// TIA Portal project "FactoryIO_Template_S7-1200_V16_V16" (V16)
// Vorlageprojekt für das Buch mit Zielsystem S7-1200

(* hardware
DEVICE "S7-1200-Station_1"  S7-1200 Station
   slot 0: "Baugruppenträger_0"  Rack  V1.0
   slot 1: "PLC_1"  CPU 1211C DC/DC/DC  6ES7 211-1AE40-0XB0  V4.1
*)

// ===== PLC "PLC_1"  CPU 1211C DC/DC/DC =====

VAR_GLOBAL   // PLC tag table "Standard-Variablentabelle"
   "Tag_4" AT %I10.0 : Bool;
   "Tag_5" AT %Q10.0 : Bool;
   "Tag_6" AT %I10.1 : Bool;
   "loop marker" AT %M0.0 : Bool;
   "Before Two Axis (-)" AT %M0.1 : Bool;
   "Tag_1" AT %M2.0 : Bool;
   "Tag_2" AT %M2.1 : Bool;
   "Tag_3" AT %M2.2 : Bool;
   "Tag_7" AT %M2.3 : Bool;
   "z-move-s1" AT %M0.2 : Bool;
   "stop x -s1" AT %M0.3 : Bool;
   "x-move-s1" AT %M0.4 : Bool;
   "rotate CC-1" AT %M0.5 : Bool;
   "rotate CCW-1" AT %M0.6 : Bool;
   "x-move-s2" AT %M0.7 : Bool;
   "z-move-s2" AT %M1.0 : Bool;
   "stop x -s2" AT %M1.1 : Bool;
   "counter reset marker" AT %M1.2 : Bool;
   "grab control" AT %M1.3 : Bool;
END_VAR

VAR_GLOBAL   // PLC tag table "Tag table from XML_1"
   "Start Button" AT %I0.0 : Bool;
   "Stop Button" AT %I0.1 : Bool;
   "low sensor" AT %I0.2 : Bool;
   "High Sensor" AT %I0.3 : Bool;
   "Before Two Axis" AT %I0.4 : Bool;
   "Two-Axis Pick & Place  (Moving X Detected)" AT %I0.5 : Bool;
   "Two-Axis Pick & Place  (Moving Z Detected)" AT %I0.6 : Bool;
   "Two-Axis Pick & Place  (Detected)" AT %I0.7 : Bool;
   "Two-Axis Pick & Place  (Rotating Detected)" AT %I1.0 : Bool;
   "Entry Conveyor" AT %Q0.0 : Bool;
   "Sorting Conveyor" AT %Q0.1 : Bool;
   "Small Conveyor" AT %Q0.2 : Bool;
   "Large Conveyor" AT %Q0.3 : Bool;
   "Two-Axis Pick & Place  (Moving X)" AT %Q0.4 : Bool;
   "Two-Axis Pick & Place  (Moving Z)" AT %Q0.5 : Bool;
   "Two-Axis Pick & Place  (Grab)" AT %Q0.6 : Bool;
   "Two-Axis Pick & Place  (Rotate CW)" AT %Q0.7 : Bool;
   "Two-Axis Pick & Place  (Rotate CCW)" AT %Q1.0 : Bool;
   "Start Button  (Light)" AT %Q1.1 : Bool;
   "Stop Button  (Light)" AT %Q1.2 : Bool;
END_VAR

// folder: System blocks/Program resources

DATA_BLOCK "movement-counter"   // DB1
{ S7_Optimized_Access := 'TRUE' }
AUTHOR : Simatic
FAMILY : IEC
NAME : CNTR
VERSION : 1.0
// stored: InstanceOfName IEC_COUNTER
"IEC_COUNTER"
BEGIN
END_DATA_BLOCK

DATA_BLOCK "grap-delay"   // DB2
{ S7_Optimized_Access := 'TRUE' }
AUTHOR : Simatic
FAMILY : IEC
NAME : IEC_TMR
VERSION : 1.0
// stored: InstanceOfName IEC_TIMER
"IEC_TIMER"
BEGIN
END_DATA_BLOCK

DATA_BLOCK "release delay"   // DB3
{ S7_Optimized_Access := 'TRUE' }
AUTHOR : Simatic
FAMILY : IEC
NAME : IEC_TMR
VERSION : 1.0
// stored: InstanceOfName IEC_TIMER
"IEC_TIMER"
BEGIN
END_DATA_BLOCK

// folder: (top level)

FUNCTION "MHJ-PLC-Lab-Function-S71200" : Void   // FC9000, SCL
{ S7_Optimized_Access := 'TRUE' }
VERSION : 0.1
   VAR_TEMP
      rdTimeReturn : Int;
      outputTime : DTL;
      SyncVal : Byte;
      forVal : Int;
      forVal_2 : Int;
      Value : Byte;
   END_VAR
   VAR CONSTANT
      CompVal : Byte := 16#34;
      Value_01 : Byte := 16#11;
      Value_01_DW : DWord := 16#A165_D992;
      Value_02_DW : DWord := 16#58BE_4401;
   END_VAR
BEGIN

   #Value:=PEEK(area := 16#82,
        dbNumber := 0,
        byteOffset := 511);
   #Value := #Value + 1;

   POKE(area := 16#82,
        dbNumber := 0,
        byteOffset := 511,
        value := #Value);

   POKE(area:=16#81,
        dbNumber:=0,
        byteOffset:=1016,
        value:=#Value_01_DW);
   POKE(area := 16#81,
        dbNumber := 0,
        byteOffset := 1020,
        value := #Value_02_DW);

   POKE(area := 16#81,
        dbNumber := 0,
        byteOffset := 511,
        value := B#16#00);

   FOR #forVal := 0 TO 120 DO
       FOR #forVal_2:=0 TO 10 DO
           #rdTimeReturn:=RD_SYS_T(#outputTime);
           #rdTimeReturn := WR_SYS_T(#outputTime);
           #rdTimeReturn := RD_SYS_T(#outputTime);
           #rdTimeReturn := WR_SYS_T(#outputTime);
       END_FOR;
       #SyncVal:= PEEK(area := 16#81,
                      dbNumber := 0,
                      byteOffset := 511);
       IF #SyncVal = #CompVal THEN
          GOTO M_1;
       END_IF;
   END_FOR;
   RETURN;

   M_1:
   POKE(area := 16#81,
        dbNumber := 0,
        byteOffset := 511,
        value := B#16#0);
END_FUNCTION

ORGANIZATION_BLOCK "Main"   // OB1, LAD, ProgramCycle
TITLE = "Main Program Sweep (Cycle)"
{ S7_Optimized_Access := 'TRUE' }
VERSION : 0.1
   VAR_INPUT
      Initial_Call : Bool;   // Initial call of this OB
      Remanence : Bool;   // =True, if remanent data are available
   END_VAR
   VAR_TEMP   // added for the SCL form of the ladder/FBD networks
      _w1 : Bool;
      _w2 : Bool;
      _w3 : Bool;
   END_VAR
BEGIN

REGION Network 1: Konnektierungsbaustein für PLC-Lab
   // Im Netzwerk 1 wird der Konnektierungsbaustein für PLC-Lab aufgerufen.
   // Dieser Aufruf darf nicht entfernt werden!
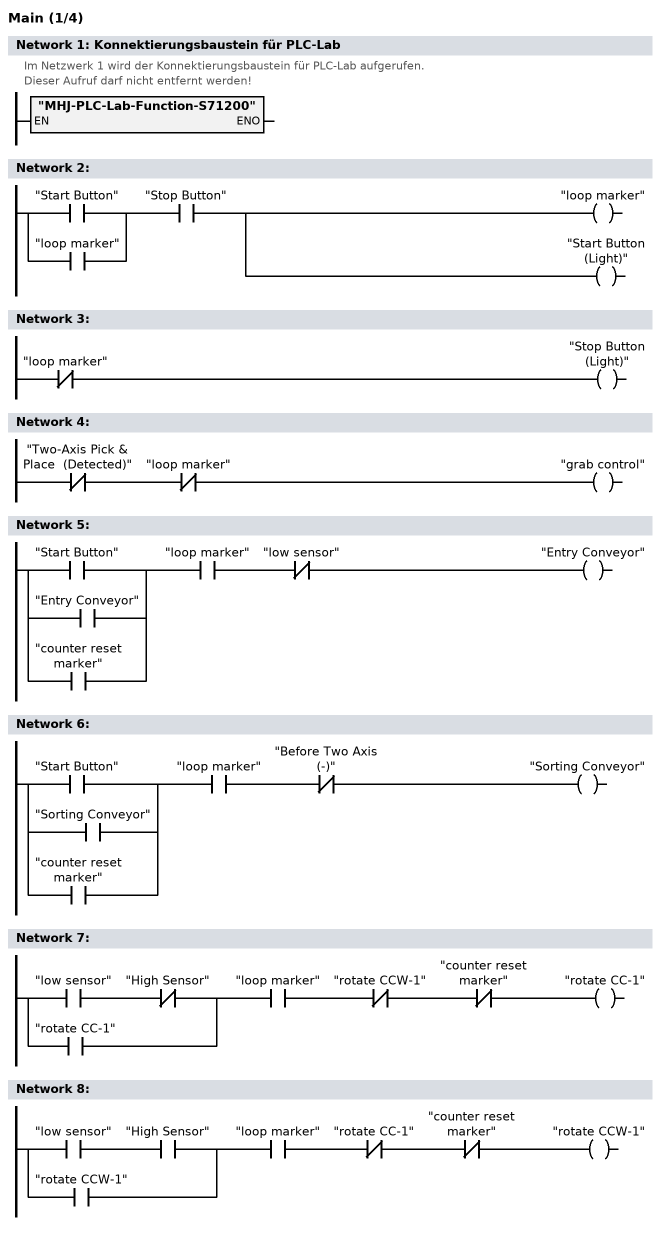
   RUNG wire#powerrail
      "MHJ-PLC-Lab-Function-S71200"()
   END_RUNG
   // the same network as SCL:
   "MHJ-PLC-Lab-Function-S71200"();
END_REGION

REGION Network 2
   RUNG wire#powerrail
      Contact( "Start Button" )
      wire#w1
      Contact( "Stop Button" )
      wire#w2
      Coil( "loop marker" )
   END_RUNG
   RUNG wire#powerrail
      Contact( "loop marker" )
   END_RUNG wire#w1
   RUNG wire#w2
      Coil( "Start Button  (Light)" )
   END_RUNG
   // the same network as SCL:
   "loop marker" := ("Start Button" OR "loop marker") AND "Stop Button";
   "Start Button  (Light)" := "loop marker";
END_REGION

REGION Network 3
   RUNG wire#powerrail
      I_Contact( "loop marker" )
      Coil( "Stop Button  (Light)" )
   END_RUNG
   // the same network as SCL:
   "Stop Button  (Light)" := NOT "loop marker";
END_REGION

REGION Network 4
   RUNG wire#powerrail
      I_Contact( "Two-Axis Pick & Place  (Detected)" )
      I_Contact( "loop marker" )
      Coil( "grab control" )
   END_RUNG
   // the same network as SCL:
   "grab control" := NOT "Two-Axis Pick & Place  (Detected)" AND NOT "loop marker";
END_REGION

REGION Network 5
   RUNG wire#powerrail
      Contact( "Start Button" )
      wire#w1
      Contact( "loop marker" )
      I_Contact( "low sensor" )
      Coil( "Entry Conveyor" )
   END_RUNG
   RUNG wire#powerrail
      Contact( "Entry Conveyor" )
   END_RUNG wire#w1
   RUNG wire#powerrail
      Contact( "counter reset marker" )
   END_RUNG wire#w1
   // the same network as SCL:
   "Entry Conveyor" := ("Start Button" OR "Entry Conveyor" OR "counter reset marker") AND "loop marker" AND NOT "low sensor";
END_REGION

REGION Network 6
   RUNG wire#powerrail
      Contact( "Start Button" )
      wire#w1
      Contact( "loop marker" )
      I_Contact( "Before Two Axis (-)" )
      Coil( "Sorting Conveyor" )
   END_RUNG
   RUNG wire#powerrail
      Contact( "Sorting Conveyor" )
   END_RUNG wire#w1
   RUNG wire#powerrail
      Contact( "counter reset marker" )
   END_RUNG wire#w1
   // the same network as SCL:
   "Sorting Conveyor" := ("Start Button" OR "Sorting Conveyor" OR "counter reset marker") AND "loop marker" AND NOT "Before Two Axis (-)";
END_REGION

REGION Network 7
   RUNG wire#powerrail
      Contact( "low sensor" )
      I_Contact( "High Sensor" )
      wire#w1
      Contact( "loop marker" )
      I_Contact( "rotate CCW-1" )
      I_Contact( "counter reset marker" )
      Coil( "rotate CC-1" )
   END_RUNG
   RUNG wire#powerrail
      Contact( "rotate CC-1" )
   END_RUNG wire#w1
   // the same network as SCL:
   "rotate CC-1" := (("low sensor" AND NOT "High Sensor") OR "rotate CC-1") AND "loop marker" AND NOT "rotate CCW-1" AND NOT "counter reset marker";
END_REGION

REGION Network 8
   RUNG wire#powerrail
      Contact( "low sensor" )
      Contact( "High Sensor" )
      wire#w1
      Contact( "loop marker" )
      I_Contact( "rotate CC-1" )
      I_Contact( "counter reset marker" )
      Coil( "rotate CCW-1" )
   END_RUNG
   RUNG wire#powerrail
      Contact( "rotate CCW-1" )
   END_RUNG wire#w1
   // the same network as SCL:
   "rotate CCW-1" := (("low sensor" AND "High Sensor") OR "rotate CCW-1") AND "loop marker" AND NOT "rotate CC-1" AND NOT "counter reset marker";
END_REGION

REGION Network 9
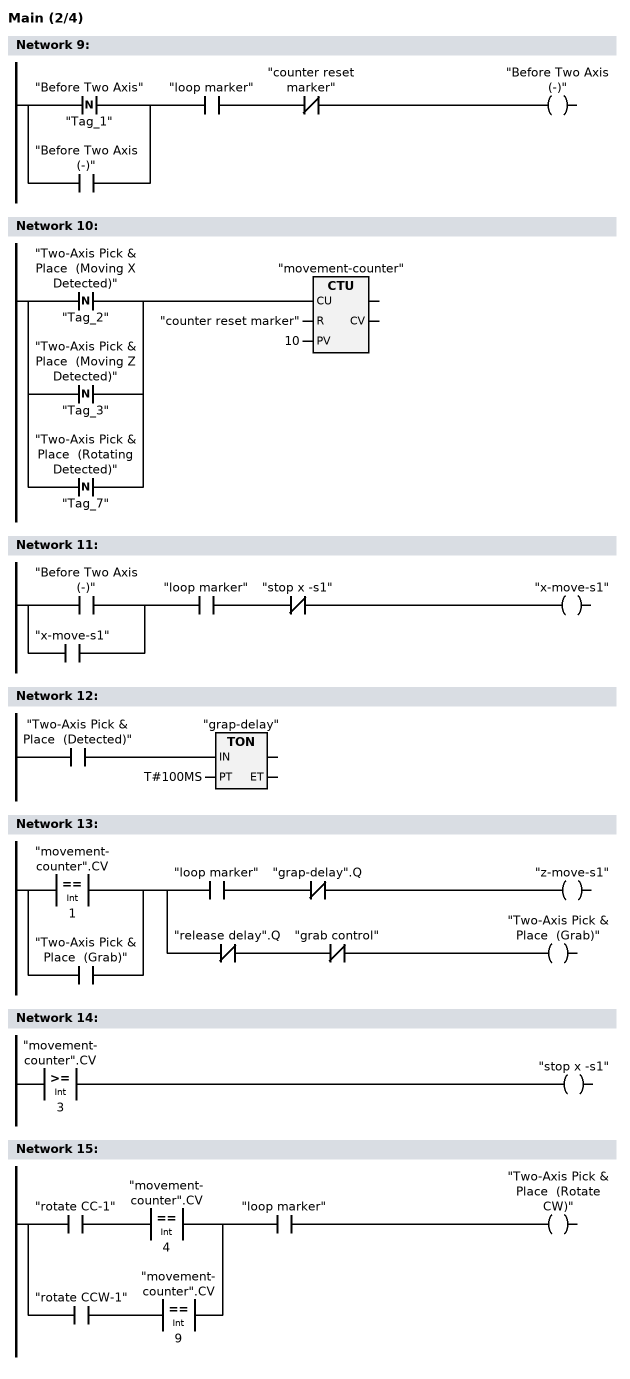
   RUNG wire#powerrail
      N_Contact(operand := "Before Two Axis", bit := "Tag_1")
      wire#w1
      Contact( "loop marker" )
      I_Contact( "counter reset marker" )
      Coil( "Before Two Axis (-)" )
   END_RUNG
   RUNG wire#powerrail
      Contact( "Before Two Axis (-)" )
   END_RUNG wire#w1
   // the same network as SCL:
   #_w1 := NOT "Before Two Axis" AND "Tag_1";   // falling edge of "Before Two Axis"
   "Tag_1" := "Before Two Axis";
   "Before Two Axis (-)" := (#_w1 OR "Before Two Axis (-)") AND "loop marker" AND NOT "counter reset marker";
END_REGION

REGION Network 10
   #_w1 := NOT "Two-Axis Pick & Place  (Moving X Detected)" AND "Tag_2";   // falling edge of "Two-Axis Pick & Place  (Moving X Detected)"
   "Tag_2" := "Two-Axis Pick & Place  (Moving X Detected)";
   #_w2 := NOT "Two-Axis Pick & Place  (Moving Z Detected)" AND "Tag_3";   // falling edge of "Two-Axis Pick & Place  (Moving Z Detected)"
   "Tag_3" := "Two-Axis Pick & Place  (Moving Z Detected)";
   #_w3 := NOT "Two-Axis Pick & Place  (Rotating Detected)" AND "Tag_7";   // falling edge of "Two-Axis Pick & Place  (Rotating Detected)"
   "Tag_7" := "Two-Axis Pick & Place  (Rotating Detected)";
   "movement-counter".CTU(CU := #_w1 OR #_w2 OR #_w3, R := "counter reset marker", PV := 10);
END_REGION

REGION Network 11
   RUNG wire#powerrail
      Contact( "Before Two Axis (-)" )
      wire#w1
      Contact( "loop marker" )
      I_Contact( "stop x -s1" )
      Coil( "x-move-s1" )
   END_RUNG
   RUNG wire#powerrail
      Contact( "x-move-s1" )
   END_RUNG wire#w1
   // the same network as SCL:
   "x-move-s1" := ("Before Two Axis (-)" OR "x-move-s1") AND "loop marker" AND NOT "stop x -s1";
END_REGION

REGION Network 12
   "grap-delay".TON(IN := "Two-Axis Pick & Place  (Detected)", PT := T#100MS);
END_REGION

REGION Network 13
   RUNG wire#powerrail
      { S7_Templates := "SrcType := Int" } EQ_Contact(in1 := "movement-counter".CV, in2 := 1)
      wire#w1
      Contact( "loop marker" )
      I_Contact( "grap-delay".Q )
      Coil( "z-move-s1" )
   END_RUNG
   RUNG wire#powerrail
      Contact( "Two-Axis Pick & Place  (Grab)" )
   END_RUNG wire#w1
   RUNG wire#w1
      I_Contact( "release delay".Q )
      I_Contact( "grab control" )
      Coil( "Two-Axis Pick & Place  (Grab)" )
   END_RUNG
   // the same network as SCL:
   #_w1 := ("movement-counter".CV = 1) OR "Two-Axis Pick & Place  (Grab)";
   "z-move-s1" := #_w1 AND "loop marker" AND NOT "grap-delay".Q;
   "Two-Axis Pick & Place  (Grab)" := #_w1 AND NOT "release delay".Q AND NOT "grab control";
END_REGION

REGION Network 14
   RUNG wire#powerrail
      { S7_Templates := "SrcType := Int" } GE_Contact(in1 := "movement-counter".CV, in2 := 3)
      Coil( "stop x -s1" )
   END_RUNG
   // the same network as SCL:
   "stop x -s1" := "movement-counter".CV >= 3;
END_REGION

REGION Network 15
   RUNG wire#powerrail
      Contact( "rotate CC-1" )
      { S7_Templates := "SrcType := Int" } EQ_Contact(in1 := "movement-counter".CV, in2 := 4)
      wire#w1
      Contact( "loop marker" )
      Coil( "Two-Axis Pick & Place  (Rotate CW)" )
   END_RUNG
   RUNG wire#powerrail
      Contact( "rotate CCW-1" )
      { S7_Templates := "SrcType := Int" } EQ_Contact(in1 := "movement-counter".CV, in2 := 9)
   END_RUNG wire#w1
   // the same network as SCL:
   "Two-Axis Pick & Place  (Rotate CW)" := (("rotate CC-1" AND ("movement-counter".CV = 4)) OR ("rotate CCW-1" AND ("movement-counter".CV = 9))) AND "loop marker";
END_REGION

REGION Network 16
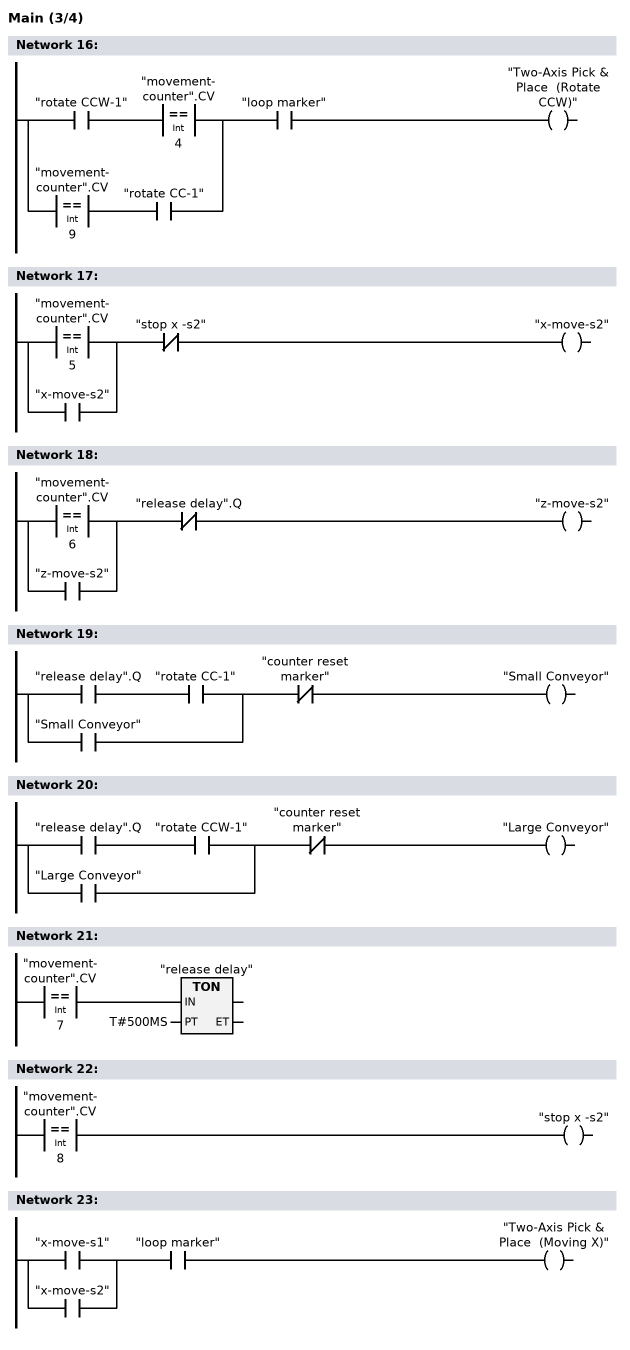
   RUNG wire#powerrail
      Contact( "rotate CCW-1" )
      { S7_Templates := "SrcType := Int" } EQ_Contact(in1 := "movement-counter".CV, in2 := 4)
      wire#w1
      Contact( "loop marker" )
      Coil( "Two-Axis Pick & Place  (Rotate CCW)" )
   END_RUNG
   RUNG wire#powerrail
      { S7_Templates := "SrcType := Int" } EQ_Contact(in1 := "movement-counter".CV, in2 := 9)
      Contact( "rotate CC-1" )
   END_RUNG wire#w1
   // the same network as SCL:
   "Two-Axis Pick & Place  (Rotate CCW)" := (("rotate CCW-1" AND ("movement-counter".CV = 4)) OR (("movement-counter".CV = 9) AND "rotate CC-1")) AND "loop marker";
END_REGION

REGION Network 17
   RUNG wire#powerrail
      { S7_Templates := "SrcType := Int" } EQ_Contact(in1 := "movement-counter".CV, in2 := 5)
      wire#w1
      I_Contact( "stop x -s2" )
      Coil( "x-move-s2" )
   END_RUNG
   RUNG wire#powerrail
      Contact( "x-move-s2" )
   END_RUNG wire#w1
   // the same network as SCL:
   "x-move-s2" := (("movement-counter".CV = 5) OR "x-move-s2") AND NOT "stop x -s2";
END_REGION

REGION Network 18
   RUNG wire#powerrail
      { S7_Templates := "SrcType := Int" } EQ_Contact(in1 := "movement-counter".CV, in2 := 6)
      wire#w1
      I_Contact( "release delay".Q )
      Coil( "z-move-s2" )
   END_RUNG
   RUNG wire#powerrail
      Contact( "z-move-s2" )
   END_RUNG wire#w1
   // the same network as SCL:
   "z-move-s2" := (("movement-counter".CV = 6) OR "z-move-s2") AND NOT "release delay".Q;
END_REGION

REGION Network 19
   RUNG wire#powerrail
      Contact( "release delay".Q )
      Contact( "rotate CC-1" )
      wire#w1
      I_Contact( "counter reset marker" )
      Coil( "Small Conveyor" )
   END_RUNG
   RUNG wire#powerrail
      Contact( "Small Conveyor" )
   END_RUNG wire#w1
   // the same network as SCL:
   "Small Conveyor" := (("release delay".Q AND "rotate CC-1") OR "Small Conveyor") AND NOT "counter reset marker";
END_REGION

REGION Network 20
   RUNG wire#powerrail
      Contact( "release delay".Q )
      Contact( "rotate CCW-1" )
      wire#w1
      I_Contact( "counter reset marker" )
      Coil( "Large Conveyor" )
   END_RUNG
   RUNG wire#powerrail
      Contact( "Large Conveyor" )
   END_RUNG wire#w1
   // the same network as SCL:
   "Large Conveyor" := (("release delay".Q AND "rotate CCW-1") OR "Large Conveyor") AND NOT "counter reset marker";
END_REGION

REGION Network 21
   "release delay".TON(IN := "movement-counter".CV = 7, PT := T#500MS);
END_REGION

REGION Network 22
   RUNG wire#powerrail
      { S7_Templates := "SrcType := Int" } EQ_Contact(in1 := "movement-counter".CV, in2 := 8)
      Coil( "stop x -s2" )
   END_RUNG
   // the same network as SCL:
   "stop x -s2" := "movement-counter".CV = 8;
END_REGION

REGION Network 23
   RUNG wire#powerrail
      Contact( "x-move-s1" )
      wire#w1
      Contact( "loop marker" )
      Coil( "Two-Axis Pick & Place  (Moving X)" )
   END_RUNG
   RUNG wire#powerrail
      Contact( "x-move-s2" )
   END_RUNG wire#w1
   // the same network as SCL:
   "Two-Axis Pick & Place  (Moving X)" := ("x-move-s1" OR "x-move-s2") AND "loop marker";
END_REGION

REGION Network 24
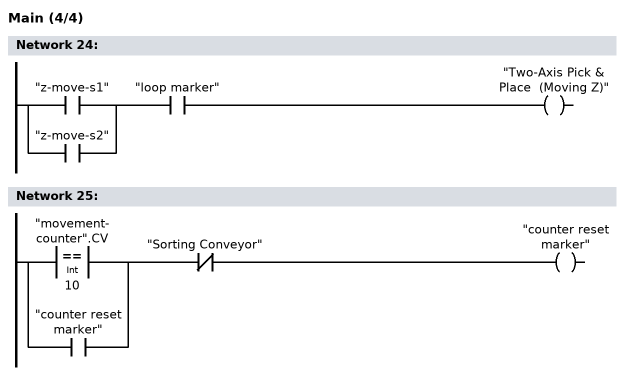
   RUNG wire#powerrail
      Contact( "z-move-s1" )
      wire#w1
      Contact( "loop marker" )
      Coil( "Two-Axis Pick & Place  (Moving Z)" )
   END_RUNG
   RUNG wire#powerrail
      Contact( "z-move-s2" )
   END_RUNG wire#w1
   // the same network as SCL:
   "Two-Axis Pick & Place  (Moving Z)" := ("z-move-s1" OR "z-move-s2") AND "loop marker";
END_REGION

REGION Network 25
   RUNG wire#powerrail
      { S7_Templates := "SrcType := Int" } EQ_Contact(in1 := "movement-counter".CV, in2 := 10)
      wire#w1
      I_Contact( "Sorting Conveyor" )
      Coil( "counter reset marker" )
   END_RUNG
   RUNG wire#powerrail
      Contact( "counter reset marker" )
   END_RUNG wire#w1
   // the same network as SCL:
   "counter reset marker" := (("movement-counter".CV = 10) OR "counter reset marker") AND NOT "Sorting Conveyor";
END_REGION
END_ORGANIZATION_BLOCK